TYPE ST_PositioningProfile :
STRUCT
	sName : STRING := 'name';
	fPosition : LREAL := 1.0;
	fVelocity : LREAL := 10.0; 
	fAcceleration : LREAL := 100.0; 
	fDeceleration : LREAL := 100.0; 
	fJerk : LREAL := 1000.0;
END_STRUCT
END_TYPE

(* stored: Version 1.1.0.1, ProductVersion 3.1.4024.12
   DUT ST_PositioningProfile: Id {83f008e9-e424-475b-ac6b-e0c4761275e2} *)
